# EPICS StreamDevice protocol: db/WFG.proto
InTerminator = LF;
OutTerminator = LF;

getId{
	out "*IDN?";
	in "%70c";
}
